{attribute 'GeneratedUsingTerminal: EL6021-0000-0016'}
{attribute addProperty BoxType "EL6021-0000-0016"}
{attribute addProperty Id "COM_InputsAT %I*COM_Inputs_3801C95E30COM_OutputsAT %Q*COM_Outputs_DEF408EC27WcStateAT %I*WcState_9091E0EB2InfoDataAT %I*InfoData_32EB74EA10"}
{attribute addProperty CRC "3046302154"}
{attribute addProperty Size "69"}
TYPE EL6021_B592E1CA EXTENDS EtcSlaveTerminalBase_947E5A46 :
STRUCT
	{attribute addProperty Name "COM_Inputs"}
	COM_Inputs : COM_Inputs_3801C95E;
	{attribute addProperty Name "COM_Outputs"}
	COM_Outputs : COM_Outputs_DEF408EC;
	{attribute addProperty Name "WcState"}
	WcState : WcState_9091E0EB;
	{attribute addProperty Name "InfoData"}
	InfoData : InfoData_32EB74EA;
END_STRUCT
END_TYPE

(* stored: Version 1.2.0.0, ProductVersion 3.1.4024.9
   DUT EL6021_B592E1CA: Id {30744b9d-dd04-4bd7-862c-5ee131ec66e8} *)
